{attribute 'qualified_only'}
{attribute 'strict'}
TYPE E_ConveyorStation :
(
	enum_member := 0
);
END_TYPE

(* stored: Version 1.1.0.1, ProductVersion 3.1.4024.12
   DUT E_ConveyorStation: Id {e5e62fa7-7dcf-4374-b53b-d59a72072455} *)
